(* Logix 5000 project; controller BallnPlate 5069-L306ERM rev 30.11; software revision 30.00 *)

TASK MainTask (periodic, rate 10 ms, priority 10, watchdog 500 ms) : MainProgram

MODULES
   Local : 5069-L306ERM (5069 0, rev 30.11)
       : 5069-IF8 (5069 3, rev 2.1, StandardDataDriven RPI 100 ms)
       : 5069-IB16 (5069 1, rev 2.1, StandardDataDriven RPI 5 ms)
       : 5069-OB16 (5069 2, rev 2.1, StandardDataDriven RPI 5 ms)
       : vendor 1 type 115 code 320 (5069 4, rev 2.1, StandardDataDriven RPI 80 ms)
END_MODULES

PROGRAM MainProgram   (* main routine Main *)
VAR
   ArduinoVoltage : DINT;
   Desired_X_Location : DINT;
   Desired_Y_Location : DINT;
   Kd : REAL;
   Kdx : REAL;
   Kix : REAL;
   Kpx : REAL;
   X_in : ALIAS FOR Local:3:I.Ch01.Data;
   X_out : ALIAS FOR Local:4:O.Ch01.Data;
   Xout : ALIAS FOR Local:4:O.Ch02.Data;
   Y_in : ALIAS FOR Local:3:I.Ch00.Data;
   Y_out : ALIAS FOR Local:4:O.Ch00.Data;
   Yout : ALIAS FOR Local:4:O.Ch00.Data;
END_VAR

ROUTINE Main   (* function block diagram *)
   SHEET 1
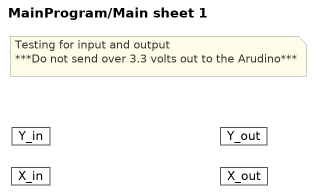
   // Testing for input and output
   // ***Do not send over 3.3 volts out to the Arudino***
   // unwired input reference Y_in
   // unwired input reference X_in
   // unwired output reference Y_out
   // unwired output reference X_out
END_ROUTINE
END_PROGRAM
